(* IEC 61131-3 sources: Industry-PLC-LLM/data/PLCBEAD_repo/PLCBEAD_PLCEmbed-main/PLC-BEAD/Source/GEB/KMH_TO_MS, 1 file *)

(* ---- KMH_TO_MS.ST ---- *)
FUNCTION KMH_TO_MS:REAL

	VAR_INPUT
		KMH :	REAL;
	END_VAR

	KMH_TO_MS := KMH * 0.2777777777777;

END_FUNCTION

PROGRAM program0
	VAR
		KMH : REAL;
		OUT : REAL;
	END_VAR

	OUT := KMH_TO_MS(KMH);
END_PROGRAM
